KUKA KRL program: chk_w2_wechs_ok.src

&ACCESS RV10
&REL 8
&COMMENT Check X1
DEF chk_w2_wechs_ok( )

; VERIFICAÇÃO DE FERRAMENTA: PINÇA X1

WAIT FOR (($IN[161]) AND ($IN[169]) AND (NOT $IN[177]) AND ($IN[185]) AND ($IN[193]) AND ($IN[219]))

END
